TYPE EL2596_Data :
STRUCT
	{attribute addProperty Name "DOX Status"}
	DOXStatus : DOXStatusChannel;
	{attribute addProperty Name "DOX Control"}
	DOXControl : DOXControlChannel;
END_STRUCT
END_TYPE

(* stored: Version 1.1.0.1, ProductVersion 3.1.4024.9
   DUT EL2596_Data: Id {86b629fb-3ad7-086c-1cae-9f92e4844fc1} *)
